{attribute 'qualified_only'}
{attribute 'strict'}
TYPE E_Status :
(
	NOTREADY,
	READY,
	STARTING,
	RUNNING,
	STOPPING,
	FAULT
);
END_TYPE

(* stored: Version 1.1.0.1, ProductVersion 3.1.4024.12
   DUT E_Status: Id {4d72eecb-d85b-47e4-b405-842ddb054f1b} *)
